(*
SPDX-FileCopyrightText: © 2026 Oleksandr Tiutyk <trofimich@gmail.com>
SPDX-License-Identifier: MIT
License: https://opensource.org/license/mit
*)

{attribute 'no_explicit_call' := 'do not call this function block directly'}
FUNCTION_BLOCK IntersectionController EXTENDS TOF_Automation.AutomationController<12> IMPLEMENTS IIntersectionController
VAR_STAT
	//! <summary>Class name shared by all instances of this function block.</summary>
	{attribute 'hide'} 
	_ClassName : STRING := __POUNAME();
END_VAR
VAR	
	{attribute 'hide'} 
	_IsOn : BOOL;
	{attribute 'hide'} 
	_FlashingYellowModeOn : BOOL;
	{attribute 'hide'} 
	_SwitchingSpeedCorrectionPercent : SPEED_CORRECTION_PERCENT;
	
	{attribute 'hide'} 
	_LightsState : INTERSECTION_LIGHTS_STATE;
	{attribute 'hide'} 
	_NextState : INTERSECTION_LIGHTS_STATE;
	
	{region "Device instances"}

	_ResetButton : TOF_Devices_IO.DigitalInput("ResetButton", THIS^);
	
	_TurnOnButton : TOF_Devices_IO.DigitalInput("TurnOnButton", THIS^);
	_TurnOffButton : TOF_Devices_IO.DigitalInput("TurnOffButton", THIS^);
	
	_SetYellowFlashingModeOnButton : TOF_Devices_IO.DigitalInput("SetYellowFlashingModeOnButton", THIS^);
	_SetYellowFlashingModeOffButton : TOF_Devices_IO.DigitalInput("SetYellowFlashingModeOffButton", THIS^);
	
	_AdjustSpeedButton : TOF_Devices_IO.DigitalInput("AdjustSpeedButton", THIS^);
	_SpeedAdjusterConverter : TOF_Devices_IO.StaticRangeAnalogValueConverter(
		minAnalogValue := -20,
		maxAnalogValue := +20,
		minRawValue := TOF_Devices_IO.RawAnalogValues.FromInt16(TOF_Core.SignedInt16.MIN_VALUE),
		maxRawValue := TOF_Devices_IO.RawAnalogValues.FromInt16(TOF_Core.SignedInt16.MAX_VALUE)
	);
	_SwitchSpeedAdjuster : TOF_Devices_IO.AnalogInput("SwitchSpeedAdjuster", THIS^, _SpeedAdjusterConverter);
	
	_TrafficLight1 : TrafficLight("TrafficLight1", THIS^);
	_TrafficLight2 : TrafficLight("TrafficLight2", THIS^);
	_TrafficLight3 : TrafficLight("TrafficLight3", THIS^);
	_TrafficLight4 : TrafficLight("TrafficLight4", THIS^);
	
	{attribute 'hide'} 	
	_DemoExceptionHandlingPolicy : DemoExceptionHandlingPolicy;
	_DemoExceptionGenerator : DemoExceptionGenerator("WatchdogDevice", THIS^);
	
 	{endregion} 	

	{region "Device related collections"}

	{attribute 'hide'} 
	_Devices : ARRAY [0.._ChildCount - 1] OF TOF_Automation.IChildAutomationComponent := 
	[
		_ResetButton,
		_TurnOnButton, 
		_TurnOffButton, 
		_SetYellowFlashingModeOnButton, 
		_SetYellowFlashingModeOffButton,
		_AdjustSpeedButton, 
		_SwitchSpeedAdjuster, 
		_TrafficLight1, 
		_TrafficLight2, 
		_TrafficLight3, 
		_TrafficLight4,
		_DemoExceptionGenerator
	];

	{attribute 'hide'} 
	_TrafficLights : ARRAY [1..IntersectionConstants.TOTAL_TRAFFIC_LIGHTS] OF ITrafficLight :=
	[
		_TrafficLight1, 
		_TrafficLight2, 
		_TrafficLight3,		
		_TrafficLight4		
	];
	{attribute 'hide'} 
	_ReadOnlyTrafficLights : POINTER TO ARRAY [1..IntersectionConstants.TOTAL_TRAFFIC_LIGHTS] OF IReadOnlyTrafficLight := ADR(_TrafficLights);
	
	{attribute 'hide'} 
	_SignalGroup1 : ARRAY [1..IntersectionConstants.TRAFFIC_LIGHTS_PER_GROUP] OF ITrafficLight :=
	[
		_TrafficLight1, 
		_TrafficLight3		
	];
	{attribute 'hide'} 
	_ReadOnlySignalGroup1 : POINTER TO
		ARRAY [1..IntersectionConstants.TRAFFIC_LIGHTS_PER_GROUP] OF IReadOnlyTrafficLight := ADR(_SignalGroup1);
	
	{attribute 'hide'} 
	_SignalGroup2 : ARRAY [1..IntersectionConstants.TRAFFIC_LIGHTS_PER_GROUP] OF ITrafficLight :=
	[
		_TrafficLight2, 
		_TrafficLight4		
	];
	{attribute 'hide'} 
	_ReadOnlySignalGroup2 : POINTER TO
		ARRAY [1..IntersectionConstants.TRAFFIC_LIGHTS_PER_GROUP] OF IReadOnlyTrafficLight := ADR(_SignalGroup2);
	
 	{endregion} 	
	
	{region "Timers"}
	
	_RedGreenLightTimer : TOF_Timers.Timer("RedGreenLightTimer");
	_YellowLightTimer : TOF_Timers.Timer("YellowLightTimer");

	_FlashingYellowLightTimer : TOF_Timers.Timer("FlashingYellowLightTimer");
	
	{endregion}
END_VAR

{attribute 'monitoring' := 'call'}
PROPERTY FINAL AdjustSpeedButton : TOF_Devices_IO.IDigitalInput
GET
AdjustSpeedButton := _AdjustSpeedButton;
END_GET
END_PROPERTY

METHOD PRIVATE bindIO
VAR
	aiChannel : POINTER TO TOF_IOModels.ANALOG_INPUT_INT_CHANNEL;
END_VAR
_ResetButton.BindToIO(
	rawValue := TerminalModels.DI_1.Ch1
);

_TurnOnButton.BindToIO(
	rawValue := TerminalModels.DI_1.Ch2
);
_TurnOffButton.BindToIO(
	rawValue := TerminalModels.DI_1.Ch3
);

_SetYellowFlashingModeOnButton.BindToIO(
	rawValue := TerminalModels.DI_1.Ch4
);
_SetYellowFlashingModeOffButton.BindToIO(
	rawValue := TerminalModels.DI_1.Ch5
);

_AdjustSpeedButton.BindToIO(
	rawValue := TerminalModels.DI_1.Ch6
);

_TrafficLight1.BindToIO(
	redLightRawValue 	:= TerminalModels.DO_2.Ch01,
	yellowLightRawValue := TerminalModels.DO_2.Ch02,
	greenLightRawValue 	:= TerminalModels.DO_2.Ch03	
);
_TrafficLight2.BindToIO(
	redLightRawValue 	:= TerminalModels.DO_2.Ch04,
	yellowLightRawValue := TerminalModels.DO_2.Ch05,
	greenLightRawValue 	:= TerminalModels.DO_2.Ch06	
);
_TrafficLight3.BindToIO(
	redLightRawValue 	:= TerminalModels.DO_2.Ch07,
	yellowLightRawValue := TerminalModels.DO_2.Ch08,
	greenLightRawValue 	:= TerminalModels.DO_2.Ch09	
);
_TrafficLight4.BindToIO(
	redLightRawValue 	:= TerminalModels.DO_2.Ch10,
	yellowLightRawValue := TerminalModels.DO_2.Ch11,
	greenLightRawValue 	:= TerminalModels.DO_2.Ch12	
);

aiChannel := ADR(TerminalModels.AI_3.Ch1);
_SwitchSpeedAdjuster.BindToInt16IO(rawValues := aiChannel^);
END_METHOD

METHOD PRIVATE calculateCorrectedInterval : TIME
VAR_INPUT
	originalInterval : TIME;
	correctionPercent : SPEED_CORRECTION_PERCENT;
END_VAR
IF correctionPercent = 0 THEN
	calculateCorrectedInterval := originalInterval;
ELSIF correctionPercent > 0 THEN
	calculateCorrectedInterval := originalInterval + TO_TIME(TO_INT(originalInterval) * correctionPercent / 100.0);
ELSE
	calculateCorrectedInterval := originalInterval - TO_TIME(TO_INT(originalInterval) * -correctionPercent / 100.0);
END_IF
END_METHOD

{attribute 'monitoring' := 'call'}
PROPERTY FINAL Children : REFERENCE TO ARRAY [0.._ChildCount - 1] OF TOF_Automation.IChildAutomationComponent
GET
Children REF= _Devices;
END_GET
END_PROPERTY

{attribute 'monitoring' := 'call'}
PROPERTY ClassName : REFERENCE TO STRING
GET
ClassName REF= _ClassName;
END_GET
END_PROPERTY

METHOD PRIVATE executeTimers
_RedGreenLightTimer.Execute();
_YellowLightTimer.Execute();
_FlashingYellowLightTimer.Execute();
END_METHOD

METHOD FB_init : BOOL
VAR_INPUT
	bInitRetains : BOOL; // TRUE: the retain variables are initialized (reset warm / reset cold)
	bInCopyCode : BOOL;  // TRUE: the instance will be copied to the copy code afterward (online change)
	name : WSTRING;
END_VAR
VAR_IN_OUT CONSTANT
	plugins : ARRAY [*] OF TOF_Automation.IAutomationControllerPlugin;
END_VAR
_DemoExceptionGenerator.ExceptionHandlingPolicy := _DemoExceptionHandlingPolicy;

AssignPlugins(plugins := plugins);
END_METHOD

{attribute 'monitoring' := 'call'}
PROPERTY FINAL LightsState : INTERSECTION_LIGHTS_STATE
GET
LightsState := _LightsState;
END_GET
END_PROPERTY

{attribute 'monitoring' := 'call'}
PROPERTY FINAL Mode : INTERSECTION_MODE
GET
IF _IsOn THEN
	Mode := SEL(_FlashingYellowModeOn, INTERSECTION_MODE.WORKING, INTERSECTION_MODE.FLASHING_YELLOW);
ELSE
	Mode := INTERSECTION_MODE.OFF;
END_IF
END_GET
END_PROPERTY

{attribute 'monitoring' := 'call'}
PROPERTY NamespaceName : REFERENCE TO STRING
GET
NamespaceName REF= CurrentNamespace.Name;
END_GET
END_PROPERTY

METHOD PROTECTED OnBeforeChildrenInitializing
_RedGreenLightTimer.Interval := IntersectionConstants.RED_GREEN_LIGHT_INTERVAL;
_YellowLightTimer.Interval := IntersectionConstants.YELLOW_LIGHT_INTERVAL;

_FlashingYellowLightTimer.Interval := IntersectionConstants.FLASHING_YELLOW_LIGHT_INTERVAL;

bindIO();
END_METHOD

METHOD PROTECTED OnBeforeChildrenStopped
IF _ResetButton.Changed AND_THEN _ResetButton.Value THEN
	Reset();
END_IF
END_METHOD

METHOD PROTECTED OnBeforeChildrenWorking
executeTimers();

IF _AdjustSpeedButton.Changed AND_THEN _AdjustSpeedButton.Value THEN
	SetSwitchingSpeedCorrectionPercent(correctionPercent := TO_SINT(_SwitchSpeedAdjuster.Value));
END_IF

IF _ResetButton.Changed AND_THEN _ResetButton.Value THEN
	Reset();
ELSIF _TurnOnButton.Changed AND_THEN _TurnOnButton.Value THEN
	TurnOn();
ELSIF _TurnOffButton.Changed AND_THEN _TurnOffButton.Value THEN
	TurnOff();
ELSIF _SetYellowFlashingModeOnButton.Changed AND_THEN _SetYellowFlashingModeOnButton.Value THEN
	SetYellowFlashingModeOn();
ELSIF _SetYellowFlashingModeOffButton.Changed AND_THEN _SetYellowFlashingModeOffButton.Value THEN
	SetYellowFlashingModeOff();
ELSE
	CASE Mode OF
		INTERSECTION_MODE.WORKING:
			processNormalMode();
		
		INTERSECTION_MODE.FLASHING_YELLOW:
			processBlinkingYellowMode();
	END_CASE
END_IF
END_METHOD

METHOD PROTECTED OnOperationalStateChanged
VAR_INPUT
	previousState : TOF_Automation.OPERATIONAL_STATE;
END_VAR
IF OperationalState = TOF_Automation.OPERATIONAL_STATE.STOPPED AND_THEN Mode <> INTERSECTION_MODE.OFF THEN
	TurnOff();
END_IF
END_METHOD

{attribute 'monitoring' := 'call'}
PROPERTY OperationalStateName : STRING(16)
GET
OperationalStateName := TO_STRING(_OperationalState);
END_GET
END_PROPERTY

METHOD PRIVATE processBlinkingYellowMode
IF _FlashingYellowLightTimer.Elapsed THEN
	IF _LightsState = INTERSECTION_LIGHTS_STATE.ALL_YELLOW THEN
		setState(
			state := INTERSECTION_LIGHTS_STATE.ALL_OFF, 
			nextState := INTERSECTION_LIGHTS_STATE.ALL_YELLOW
		);		
	ELSE
		setState(
			state := INTERSECTION_LIGHTS_STATE.ALL_YELLOW, 
			nextState := INTERSECTION_LIGHTS_STATE.ALL_OFF
		);		
	END_IF
	
	startFlashingYellowLightTimer();
	
	updateTraficLights();
END_IF
END_METHOD

METHOD processNormalMode
CASE _LightsState OF
	INTERSECTION_LIGHTS_STATE.GROUP1_GREEN_GROUP2_RED:
		IF _RedGreenLightTimer.Elapsed THEN
			startYellowLightTimer();
			
			setState(
				state := INTERSECTION_LIGHTS_STATE.ALL_YELLOW, 
				nextState := INTERSECTION_LIGHTS_STATE.GROUP1_RED_GROUP2_GREEN
			);
			
			updateTraficLights();
		END_IF
	
	INTERSECTION_LIGHTS_STATE.GROUP1_RED_GROUP2_GREEN:
		IF _RedGreenLightTimer.Elapsed THEN
			startYellowLightTimer();
			
			setState(
				state := INTERSECTION_LIGHTS_STATE.ALL_YELLOW, 
				nextState := INTERSECTION_LIGHTS_STATE.GROUP1_GREEN_GROUP2_RED
			);
			
			updateTraficLights();
		END_IF
	
	INTERSECTION_LIGHTS_STATE.ALL_YELLOW:
		IF _YellowLightTimer.Elapsed THEN
			startRedGreenLightTimer();
			
			setState(
				state := _NextState, 
				nextState := INTERSECTION_LIGHTS_STATE.ALL_YELLOW
			);
			
			updateTraficLights();
		END_IF
END_CASE
END_METHOD

{attribute 'monitoring' := 'call'}
PROPERTY FINAL ResetButton : TOF_Devices_IO.IDigitalInput
GET
ResetButton := _ResetButton;
END_GET
END_PROPERTY

{attribute 'monitoring' := 'call'}
PROPERTY SelfSize : ULINT
GET
SelfSize := XSIZEOF(THIS^);
END_GET
END_PROPERTY

METHOD INTERNAL setState
VAR_INPUT
	state : INTERSECTION_LIGHTS_STATE;
	nextState : INTERSECTION_LIGHTS_STATE;
END_VAR
_LightsState := state;
_NextState := nextState;
END_METHOD

METHOD SetSwitchingSpeedCorrectionPercent
VAR_INPUT
	correctionPercent : SPEED_CORRECTION_PERCENT;
END_VAR
_SwitchingSpeedCorrectionPercent := correctionPercent;
END_METHOD

METHOD PRIVATE setTrafficLigtsColor
VAR_IN_OUT CONSTANT
	trafficLights : ARRAY [*] OF ITrafficLight;
END_VAR
VAR_INPUT
	light : TRAFFIC_LIGHT_COLOR;
END_VAR
VAR
	i : DINT;
	
	rejectReason : WSTRING(255);
END_VAR
FOR i := LOWER_BOUND(trafficLights, 1) TO UPPER_BOUND(trafficLights, 1) DO
	IF NOT trafficLights[i].TrySetLight(color := light, rejectReason := rejectReason) THEN				
		TOF_Core.LogManager.TryLogMessage(
			message := rejectReason,
			category := TOF_Core.LOG_CATEGORY.INFORMATION,
			topic1 := TO_WSTRING(ClassName),
			topic2 := TO_WSTRING(__POUNAME()),
			topic3 := "ActionPermissionDenied"
		);
	END_IF
END_FOR
END_METHOD

METHOD SetYellowFlashingModeOff
starMode(
	isOn := _IsOn,
	flashingYellowModeOn := FALSE
);
END_METHOD

{attribute 'monitoring' := 'call'}
PROPERTY FINAL SetYellowFlashingModeOffButton : TOF_Devices_IO.IDigitalInput
GET
SetYellowFlashingModeOffButton := _SetYellowFlashingModeOffButton;
END_GET
END_PROPERTY

METHOD SetYellowFlashingModeOn
starMode(
	isOn := _IsOn,
	flashingYellowModeOn := TRUE
);
END_METHOD

{attribute 'monitoring' := 'call'}
PROPERTY FINAL SetYellowFlashingModeOnButton : TOF_Devices_IO.IDigitalInput
GET
SetYellowFlashingModeOnButton := _SetYellowFlashingModeOnButton;
END_GET
END_PROPERTY

{attribute 'monitoring' := 'call'}
PROPERTY FINAL SignalGroup1 : REFERENCE TO
	ARRAY [1..IntersectionConstants.TRAFFIC_LIGHTS_PER_GROUP] OF IReadOnlyTrafficLight
GET
SignalGroup1 REF= _ReadOnlySignalGroup1^;
END_GET
END_PROPERTY

{attribute 'monitoring' := 'call'}
PROPERTY FINAL SignalGroup2 : REFERENCE TO
	ARRAY [1..IntersectionConstants.TRAFFIC_LIGHTS_PER_GROUP] OF IReadOnlyTrafficLight
GET
SignalGroup2 REF= _ReadOnlySignalGroup2^;
END_GET
END_PROPERTY

METHOD PRIVATE starMode
VAR_INPUT
	isOn : BOOL;
	flashingYellowModeOn : BOOL;
END_VAR
_RedGreenLightTimer.Cancel();
_YellowLightTimer.Cancel();
_FlashingYellowLightTimer.Cancel();

_IsOn := isOn;
_FlashingYellowModeOn := flashingYellowModeOn;

CASE Mode OF
	INTERSECTION_MODE.OFF:
		_LightsState := INTERSECTION_LIGHTS_STATE.ALL_OFF;

	INTERSECTION_MODE.WORKING:
		startRedGreenLightTimer();
		_LightsState := INTERSECTION_LIGHTS_STATE.GROUP1_GREEN_GROUP2_RED;
	
	INTERSECTION_MODE.FLASHING_YELLOW:
		_LightsState := INTERSECTION_LIGHTS_STATE.ALL_YELLOW;
		startFlashingYellowLightTimer();
END_CASE

updateTraficLights();
END_METHOD

METHOD PRIVATE startFlashingYellowLightTimer

_FlashingYellowLightTimer.Interval := calculateCorrectedInterval(
	originalInterval := IntersectionConstants.FLASHING_YELLOW_LIGHT_INTERVAL,
	correctionPercent := _SwitchingSpeedCorrectionPercent
);

_FlashingYellowLightTimer.Restart();
END_METHOD

METHOD PRIVATE startRedGreenLightTimer

_RedGreenLightTimer.Interval := calculateCorrectedInterval(
	originalInterval := IntersectionConstants.RED_GREEN_LIGHT_INTERVAL,
	correctionPercent := _SwitchingSpeedCorrectionPercent
);

_RedGreenLightTimer.Restart();
END_METHOD

METHOD PRIVATE startYellowLightTimer

_YellowLightTimer.Interval := calculateCorrectedInterval(
	originalInterval := IntersectionConstants.YELLOW_LIGHT_INTERVAL,
	correctionPercent := _SwitchingSpeedCorrectionPercent
);

_YellowLightTimer.Restart();
END_METHOD

{attribute 'monitoring' := 'call'}
PROPERTY FINAL SwitchingSpeedCorrectionPercent : SINT(-20..+20)
GET
SwitchingSpeedCorrectionPercent := _SwitchingSpeedCorrectionPercent;
END_GET
END_PROPERTY

{attribute 'monitoring' := 'call'}
PROPERTY FINAL SwitchSpeedAdjuster : TOF_Devices_IO.IAnalogInput
GET
SwitchSpeedAdjuster := _SwitchSpeedAdjuster;
END_GET
END_PROPERTY

METHOD ThrowExceptionInDemoExceptionGenerator
VAR_IN_OUT CONSTANT
	exceptionMessage : STRING(255);
	isCritical : BOOL; 
END_VAR
_DemoExceptionGenerator.ThrowException(exceptionMessage := exceptionMessage, isCritical := isCritical);
END_METHOD

{attribute 'monitoring' := 'call'}
PROPERTY FINAL TrafficLights : REFERENCE TO ARRAY [1..IntersectionConstants.TOTAL_TRAFFIC_LIGHTS] OF IReadOnlyTrafficLight
GET
TrafficLights REF= _ReadOnlyTrafficLights^;
END_GET
END_PROPERTY

METHOD TurnOff
starMode(
	isOn := FALSE,
	flashingYellowModeOn := _FlashingYellowModeOn
);
END_METHOD

{attribute 'monitoring' := 'call'}
PROPERTY FINAL TurnOffButton : TOF_Devices_IO.IDigitalInput
GET
TurnOffButton := _TurnOffButton;
END_GET
END_PROPERTY

METHOD TurnOn
starMode(
	isOn := TRUE,
	flashingYellowModeOn := _FlashingYellowModeOn
);
END_METHOD

{attribute 'monitoring' := 'call'}
PROPERTY FINAL TurnOnButton : TOF_Devices_IO.IDigitalInput
GET
TurnOnButton := _TurnOnButton;
END_GET
END_PROPERTY

METHOD PRIVATE updateTraficLights
CASE _LightsState OF
	INTERSECTION_LIGHTS_STATE.ALL_OFF:
		setTrafficLigtsColor(trafficLights := _TrafficLights, light := TRAFFIC_LIGHT_COLOR.NO_COLOR);
	
	INTERSECTION_LIGHTS_STATE.ALL_YELLOW:
		setTrafficLigtsColor(trafficLights := _TrafficLights, light := TRAFFIC_LIGHT_COLOR.YELLOW);
	
	INTERSECTION_LIGHTS_STATE.GROUP1_GREEN_GROUP2_RED:
		setTrafficLigtsColor(trafficLights := _SignalGroup1, light := TRAFFIC_LIGHT_COLOR.GREEN);
		setTrafficLigtsColor(trafficLights := _SignalGroup2, light := TRAFFIC_LIGHT_COLOR.RED);
	
	INTERSECTION_LIGHTS_STATE.GROUP1_RED_GROUP2_GREEN:
		setTrafficLigtsColor(trafficLights := _SignalGroup1, light := TRAFFIC_LIGHT_COLOR.RED);
		setTrafficLigtsColor(trafficLights := _SignalGroup2, light := TRAFFIC_LIGHT_COLOR.GREEN);
END_CASE
END_METHOD

END_FUNCTION_BLOCK

(* stored: Version 1.1.0.1
   POU IntersectionController: Id {d0f0aa39-ea76-461a-8fa3-dba15b8635a6}, SpecialFunc None
   Folder Commands: Id {f2e82d7a-5ab5-47e6-a7c7-dc6438a69b54}
   Folder Overriden methods: Id {13702960-9d99-4885-a6ce-63462aae1b07}
   Folder Service methods: Id {856d71ee-39f1-4125-9914-d1908aaa9de4}
   Folder Process mode: Id {9df05ec4-b756-4783-a76b-40e885978be7}
   Folder Start timer: Id {c16a13e4-4c94-4831-b2dc-b8960e14f551}
   Folder Statuses: Id {085c842a-347d-4cc3-8235-05f6d74ef9e6}
   Folder Subdevices: Id {710d8326-d80e-4952-8d13-0738681ba94c}
   Property AdjustSpeedButton: Id {0e8de7ff-e0de-4178-bb7b-65c754591901}
   Get Get: Id {dead62fc-07a9-4404-83ab-c23a9824c993}
   Method bindIO: Id {1bc433ca-8d0e-4452-8e3c-75449de42a8a}
   Method calculateCorrectedInterval: Id {51d751ca-80fc-4362-91e8-31296f350aff}
   Property Children: Id {edb09d7e-eaa4-4ee7-bf71-f499880b4098}
   Get Get: Id {90a76f6a-9caa-4ca6-88e8-931aff742de9}
   Property ClassName: Id {533645c9-51ab-4278-b915-2be070529db7}
   Get Get: Id {1aae8f98-7140-4915-9ec0-3cdf6e26caf7}
   Method executeTimers: Id {dfed4c3f-27bc-4f55-8a83-85a2d79b2492}
   Method FB_init: Id {cc48a528-d8b0-42ce-9f2b-4916737cac09}
   Property LightsState: Id {0d41ded4-f538-4005-aa70-f221d58f38a5}
   Get Get: Id {7519eabe-1cc3-4af8-82b3-a2f8425fe098}
   Property Mode: Id {70c7bc2d-0923-4507-922c-273224e7708a}
   Get Get: Id {0c285f66-f61a-47a3-955f-b140c5836c96}
   Property NamespaceName: Id {b7a7d419-b6f1-4dfe-b4b4-ae9ac4b21e47}
   Get Get: Id {225fc0aa-c40a-4b1c-a5e5-ec5ea749c036}
   Method OnBeforeChildrenInitializing: Id {d14266f5-308f-4ec2-bbd3-dd4787db6449}
   Method OnBeforeChildrenStopped: Id {0516e5db-6b58-48f7-b149-9edab8091cfe}
   Method OnBeforeChildrenWorking: Id {a2091fd1-b3c2-4408-9e2a-b795dd68dcf8}
   Method OnOperationalStateChanged: Id {dfa58b81-4624-4688-b85b-fa55f112c836}
   Property OperationalStateName: Id {af99d547-78da-4f00-96bd-32d0d0304681}
   Get Get: Id {7a068cfa-95a9-4134-b604-ea1c07f183d2}
   Method processBlinkingYellowMode: Id {62fb35a3-197f-483b-a168-1d68d2c02c71}
   Method processNormalMode: Id {a778b296-2e19-469e-8475-30ab670a6dcd}
   Property ResetButton: Id {17258f9f-04a6-4026-9d49-4d1d3b2cf340}
   Get Get: Id {2fcfe820-b683-4e4c-ba46-821a27b852e2}
   Property SelfSize: Id {db85e590-8997-4b56-bd9a-8e5dd4df70fe}
   Get Get: Id {f6ab4eca-dad6-4656-bd85-433d2bf1854b}
   Method setState: Id {5c2f2c55-d0ba-4b8a-8df7-9cfa51071236}
   Method SetSwitchingSpeedCorrectionPercent: Id {ce93f60b-ebdf-4524-8da1-82b6d19e82c7}
   Method setTrafficLigtsColor: Id {32bd3844-8f88-48f3-a224-ac959493d17c}
   Method SetYellowFlashingModeOff: Id {a46b1b82-4335-41d5-8b6c-822f10afe1d7}
   Property SetYellowFlashingModeOffButton: Id {277109e0-167c-4f25-8caa-2f4a2c1254c7}
   Get Get: Id {a4d0fca5-b801-417e-86fd-d6ab425535e8}
   Method SetYellowFlashingModeOn: Id {a8d74869-0985-48ce-8ed9-f193f84d16fd}
   Property SetYellowFlashingModeOnButton: Id {a4a71e1a-5dc0-41c8-b6e2-0a340d126fcd}
   Get Get: Id {35f9ad22-fa01-46e2-a2ae-83a8496cef6a}
   Property SignalGroup1: Id {4843127a-b5f8-4288-9d56-ada883c49d57}
   Get Get: Id {1a4eb1b3-0819-4585-b390-ed321667e91d}
   Property SignalGroup2: Id {ecc07983-e080-4dca-9104-b4c59dd18f5a}
   Get Get: Id {8facf4b3-e9c7-4a51-887f-6cbb040d8e61}
   Method starMode: Id {8ddb5609-6544-4dcc-b972-500abb23f0f5}
   Method startFlashingYellowLightTimer: Id {96309d45-677b-4977-9f1c-e21c0143efbb}
   Method startRedGreenLightTimer: Id {50f36714-64fe-4212-afb9-2e8a39734cfd}
   Method startYellowLightTimer: Id {75f70f4d-af10-457d-91be-f1022c3b5646}
   Property SwitchingSpeedCorrectionPercent: Id {514a1e2b-b7f4-43e3-8b7a-0937fa2a6efe}
   Get Get: Id {b0f07301-bd56-4f28-826e-8661c7ca988f}
   Property SwitchSpeedAdjuster: Id {06dddc90-cb5c-4f31-9411-86ecae41141b}
   Get Get: Id {af2782fd-129d-48e7-9c55-29dba0d016f0}
   Method ThrowExceptionInDemoExceptionGenerator: Id {f31810e7-aba6-420d-a3fd-5fbe3bd1cd33}
   Property TrafficLights: Id {1eb64023-b212-4c31-8a8b-6a8402e94081}
   Get Get: Id {d43f39e5-1277-4211-984b-d6561c34e197}
   Method TurnOff: Id {810e2a8d-5a15-4847-a93d-4ffb0fa45a73}
   Property TurnOffButton: Id {0d436a4c-a870-49f7-96c2-6da72c80e238}
   Get Get: Id {94182c5c-e238-4644-8fe4-20178014c768}
   Method TurnOn: Id {7a7d5ebb-876c-475e-adf9-9517420ae539}
   Property TurnOnButton: Id {c6426b4a-cc28-41ca-ab55-394b24ab5039}
   Get Get: Id {2f3df52f-dc14-4983-9392-94054660fe17}
   Method updateTraficLights: Id {f60cca55-65f4-4222-8c1f-0c67e0a9c589} *)
